SUBAPPLICATION Uebung_245_AX (* Sollwert mit festem Korrekturfaktor skalieren (AR_MUL_2 + initval_AR) - Lastteiler-Kompensation, I3 nach N3 *)
  (* Standard: 61499-2; Description: Copyright (c) 2026 Meisterschulen am Ostbahnhof This program and the accompanying materials are made available under the terms of the Eclipse Public License 2.0 which is available at https://www.eclipse.org/legal/epl-2.0/ SPDX-License-Identifier: EPL-2.0 *)
  (* Version 1.0, 2026-09-07, Franz Höpfinger, Meisterschulen am Ostbahnhof, initial API and implementation and/or initial documentation *)
  PACKAGE Uebungen;
  IMPORT Uebungen::const::UT::DefaultPool_Numeric::InputNumber_I3_N;
  IMPORT Uebungen::const::UT::DefaultPool_Numeric::OutputNumber_N3_N;
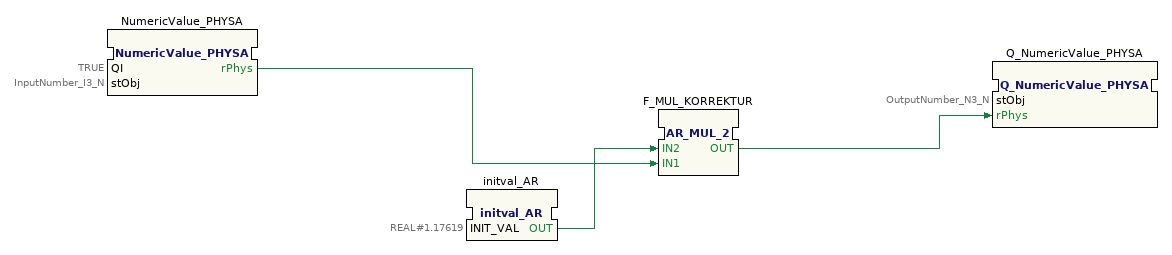
  (* Korrekturfaktor 1,17619 = 1 / 0,8502: kompensiert einen Lastteiler (z.B. PWM-Tiefpassfilter, dessen Ausgangsimpedanz gegen die Eingangsimpedanz des angeschlossenen Verbrauchers belastet wird - siehe PVEA-Kompensationsrechnung). I3 = unkorrigierter Sollwert 0-100%, N3 = korrigierter Wert, der am unbelasteten Ausgang eingestellt werden muss, damit am Verbraucher der ursprüngliche Sollwert ankommt. *)
  FBS
    NumericValue_PHYSA : isobus::UT::io::NumericValue::NumericValue_PHYSA(QI := TRUE, stObj := InputNumber_I3_N);
    F_MUL_KORREKTUR : adapter::iec61131::arithmetic::AR_MUL_2;
    Q_NumericValue_PHYSA : isobus::UT::Q::Q_NumericValue_PHYSA(stObj := OutputNumber_N3_N);
    initval_AR : adapter::types::unidirectional::AR::initval::initval_AR(INIT_VAL := REAL#1.17619);
  END_FBS
  ADAPTER_CONNECTIONS
    F_MUL_KORREKTUR.OUT TO Q_NumericValue_PHYSA.rPhys;
    initval_AR.OUT TO F_MUL_KORREKTUR.IN2;
    NumericValue_PHYSA.rPhys TO F_MUL_KORREKTUR.IN1;
  END_CONNECTIONS
END_SUBAPPLICATION
